PROGRAM MAIN
VAR
	bAllDone					: BOOL;
	bStopSequence				: BOOL;
	                    		
	nCase 						: INT;
	nMoveState				  	: ARRAY[GC.nNumMinMovers..GC.nNumMaxMovers] OF INT;
	                    		
	fbXtsEnvironment			: Tc3_XTS_Utility.FB_TcIoXtsEnvironment;
	                    		
	nForCounter					: UDINT;
	M,N,T,Tr					: UDINT;
	dynamics				    : INT;

//Status
	xSimulation					: BOOL := TRUE;
	SystemEnabled				: BOOL;

	IsMoverInBlockingArea		: BOOL;
	nActStopPos					: UINT := 1;
	Fp_error 					: Tc2_Standard.R_TRIG;
	FaultReset					: Tc2_Standard.R_TRIG;
	MoverStop 	AT%I* 			: BOOL;
    ResetSafetyLight AT%Q*      : BOOL;
	MoverStopDone AT%Q*			: BOOL;
	Info 		AT%Q*			: BOOL;
	Operating	AT%Q*			: BOOL;
	Process		AT%Q*			: BOOL;
	Fault		AT%Q*			: BOOL;
	Emergency	AT%Q*			: BOOL;
	                        	
	Voltage1	AT%I*			: UDINT;
	Voltage2	AT%I*			: UDINT;
	                        	
	TcRestart 					: Tc2_Utilities.TC_Restart;
	Restart 					: BOOL;
	busy 						: BOOL;
	fp_start 					: Tc2_Standard.R_TRIG;
	bStartSequence				: BOOL;
	                        	
	Horntimer 					: Tc2_Standard.TP; 
	R_trigHorn 					: Tc2_Standard.R_TRIG;

	StopTime 					: TIME := T#1S;
	StopTimer 					: ARRAY[GC.nNumMinMovers..GC.nNumMaxMovers] OF Tc2_Standard.TON;
	StartTimer 					: ARRAY[GC.nNumMinMovers..GC.nNumMaxMovers] OF BOOL;

	ArcLength 					: ARRAY[GC.nNumMinMovers..GC.nNumMaxMovers] OF LREAL;
	TrackPos					: ARRAY[GC.nNumMinMovers..GC.nNumMaxMovers] OF ARRAY[GC.nNumMinTracks..GC.nNumMaxTracks] OF Tc3_Physics.PositionXYC;
END_VAR

fbXtsEnvironment.Init(bExecute := TRUE);
//Cyclic
M_WritePlanarTrackConfig();
M_UpdateConfigurations();
IF xSimulation THEN
	SystemEnabled	:= TRUE;
ELSE
	SystemEnabled	:= (MoverStop (* SafetyOK *) AND NOT Fault);
END_IF

//Command Diverting to Magnet for any designated mover
DivertQueue();
HistoryDivertQueue(); // no removal
MergeQueue();

SwitchMagnet(SafetyPermIntlk := SystemEnabled,
			stSwitchConfig := GVL_General.stSwitchConfig);

Emergency :=  MoverStop;
ResetSafetyLight    := NOT MoverStop;

Operating := NOT  MoverStop;
R_trigHorn(clk := Voltage1> 10000 OR Voltage2 >10000);
Horntimer(in:= ( R_trigHorn.Q ) , PT:= T#2S,Q=> info);

IF nCase > 90 THEN
	Process := TRUE;
ELSE 
	Process := FALSE;	
END_IF

IF NOT fbXtsEnvironment.P_IsInitialized THEN
	RETURN;
END_IF

IF NOT MoverStop AND NOT MoverStopDone THEN
	FOR nForCounter:=1 TO nNumMovers DO
		aDynamics[nForCounter].SetValuesVADJ(V := stMoverConfig.MaxVelo, A := stMoverConfig.MaxAccel, D := stMoverConfig.MaxDecel, J := stMoverConfig.MaxJerk);
		nCase := 140;
		//fbPlanarMover[nForCounter].McPlanarMover.Halt(MoverFeedback[nForCounter], aDynamics[nForCounter]);
	END_FOR		
	MoverStopDone := TRUE;
ELSIF MoverStop THEN
	MoverStopDone := FALSE;
END_IF


TcRestart(
NETID:= '', 
RESTART:= Restart, 
TMOUT:=T#5S , 
BUSY=>busy , 
ERR=> , 
ERRID=> );


fp_start(CLK := bStartSequence);
IF fp_start.Q THEN
	nCase := 10;
	bStartSequence := FALSE;
END_IF

//IsMoverCommandedInShortcut := FALSE;
IsMoverInBlockingArea := FALSE;

	bAllDone:= TRUE;
FOR M := GC.nNumMinMovers TO nNumMovers DO///Movers
	StopTimer[M](in:=StartTimer[m],PT:=StopTime);
	GVL_Mc3.fbPlanarXtsMover[M].P_MoverId := M;
	GVL_Mc3.fbPlanarXtsMover[M].P_PlanarMover.MoverNumber	:= GVL_Mc3.fbPlanarXtsMover[M].nMoverId;
  GVL_Mc3.aiXpuXtsMover[M]  := fbXtsEnvironment.XpuTcIo(1).MoverTcIo(TO_UINT(M));
  fbPlanarXtsMover[M].iTcIoXtsXpuMover REF= GVL_Mc3.aiXpuXtsMover[M];
	fbPlanarXtsMover[M].Update();
	
	//MoverPos[M].SetValuesXYC(fbPlanarMover[M].McPlanarMover.MCTOPLC.SET.SetPos.x, fbPlanarMover[M].McPlanarMover.MCTOPLC.SET.SetPos.y,fbPlanarMover[M].McPlanarMover.MCTOPLC.SET.SetPos.c);
	
	TR := Tr+1;
	IF Tr = 4 THEN
		Tr :=1;
	END_IF
	{warning <'MoverPhysics does not work'>}
	ArcLength[M] :=GVL_Mc3.MC_Tracks[Tr].GetArcLengthClosestTo(GVL_Mc3.fbPlanarXtsMover[M].P_MoverPhysics);
	GVL_Mc3.MC_Tracks[Tr].GetPositionAt(ArcLength[M],TrackPos[M][Tr]);
	
//	IF ABS(GVL_Mc3.fbPlanarXtsMover[M].MoverPhysics.x - TrackPos[M][Tr].x) < 1 AND  ABS(fbPlanarXtsMover[M].MoverPhysics.y - TrackPos[M][Tr].y) < 1 THEN
// 		GVL_Mc3.fbPlanarXtsMover[M].P_XPlanarMover.MoverTrackNr := Tr;
//	END_IF	
	
//	IsMoverCommandedInShortcut := IsMoverCommandedInShortcut OR fbPlanarXtsMover[M].IsCommandedInShortcut;
//	IsMoverInBlockingArea := IsMoverInBlockingArea OR (GVL_Mc3.fbPlanarXtsMover[M].P_PlanarMover.TrackID = GVL_Mc3.MC_Tracks[E_TrackNum.main].MCTOPLC_STD.TrackOID AND 
//														IsBetween(value := GVL_Mc3.fbPlanarXtsMover[M].P_PlanarMover.MoverPos, 
//														minV := GVL_General.stSwitchConfig.fMagnetEntryPosn - GVL_General.stSwitchConfig.MagnetPosnComp, 
//														maxV :=  GVL_General.stSwitchConfig.fMagnetExitPosn + stSwitchConfig.MagnetPosnComp));
	MoverFeedback[M].Update();
	

	Fp_error(CLK := fbPlanarXtsMover[M].McPlanarMover.Error AND nCase = 100);
	IF Fp_error.Q THEN
		nCase := 140;
		Fault := TRUE;
//		bCmdMagnetOn := FALSE;
	END_IF
END_FOR

FOR T := GC.nNumMinTracks TO GC.nNumMaxTracks DO 
	MC_Tracks[T].Update();
	MC_Trackfeedback[T].Update();
END_FOR

CASE nCase OF
	10:
		Fault := FALSE;
		FOR nForCounter := 1 TO fbXtsEnvironment.XpuTcIo(1).GetPartCount() DO
			fbXtsEnvironment.XpuTcIo(1).PartTcIo(TO_UINT(nForCounter)).TriggerReset();
		END_FOR
		
		nCase := 20;

	20:
		FOR T := GC.nNumMinTracks TO GC.nNumMaxTracks DO 
			MC_Tracks[T].Enable(MC_Trackfeedback[T]);
		END_FOR
				nCase := 30;
		
		
	30: 
		IF MC_Trackfeedback[E_TrackNum.Big].Done AND MC_Trackfeedback[E_TrackNum.Main].Done AND MC_Trackfeedback[E_TrackNum.Small].Done THEN
			nCase := 35;
		END_IF
		
		
	35:
		FOR nForCounter:=GC.nNumMinMovers TO GVL_General.nNumMovers DO
			fbPlanarXtsMover[nForCounter].McPlanarMover.Reset(MoverFeedback[nForCounter]);
		END_FOR
		nCase := 36;	
		
		
	36:	
		bAllDone:=TRUE;
		FOR nForCounter:=GC.nNumMinMovers TO GVL_General.nNumMovers DO
			bAllDone:=bAllDone AND MoverFeedback[nForCounter].Done;
		END_FOR
		
		IF bAllDone THEN
			nCase := 40;
		END_IF
		
		
	40:
		FOR nForCounter:=GC.nNumMinMovers TO GVL_General.nNumMovers DO
			fbPlanarXtsMover[nForCounter].McPlanarMover.Enable(MoverFeedback[nForCounter]);
		END_FOR
		nCase := 50;
	
		
	50:
		bAllDone:=TRUE;
		FOR nForCounter:=GC.nNumMinMovers TO GVL_General.nNumMovers DO
			bAllDone:=bAllDone AND MoverFeedback[nForCounter].Done;
		END_FOR
		
		IF bAllDone THEN
			nCase := 60;
		END_IF

	//55:

	60:
		FOR nForCounter:=GC.nNumMinMovers TO GVL_General.nNumMovers DO
			IF nForCounter <= 9 THEN
				fbPlanarXtsMover[nForCounter].JoinTrack(MoverFeedback[nForCounter], GVL_Mc3.MC_Tracks[E_TrackNum.Big]);//   Mover[nForCounter].MoverTrackNr]);
			ELSE
				fbPlanarXtsMover[nForCounter].JoinTrack(MoverFeedback[nForCounter], GVL_Mc3.MC_Tracks[E_TrackNum.Main]);
			END_IF	
		END_FOR
		
		nCase := 70;
		
	70:
		bAllDone:=TRUE;
		FOR nForCounter:=GC.nNumMinMovers TO GVL_General.nNumMovers DO
			bAllDone:=bAllDone AND MoverFeedback[nForCounter].Done;
		END_FOR
		
		IF bAllDone THEN
			nCase := 80;
		END_IF
		
	80:	
		FOR nForCounter:=GC.nNumMinMovers TO GVL_General.nNumMovers DO
			nMoveState[nForCounter] := 0;
			aMoveOnTrackOptions[nForCounter].direction := MC_Direction.mcDirectionPositive;
			aMoveOnTrackOptions[nForCounter].gapMode := MC_GAP_MODE_ON_TRACK.Fast1D;
		END_FOR
		
		nCase := 100;

	100:

		FOR nForCounter:= GC.nNumMinMovers TO GVL_General.nNumMovers DO
			IF TrackSectors[nForCounter].SectorStatus[GC.SHORTCUT_HD_SECTION].MoverIsOnSector THEN
				//Increase dynamics on Inner Shortcut
				aDynamics[nForCounter].SetValuesVADJ(V := stMoverConfig.NormalVelo, A := stMoverConfig.MaxAccel, D := stMoverConfig.MaxDecel, J := stMoverConfig.MaxJerk);
//				aMoveOnTrackOptions[nForCounter].gap:= stMoverConfig.TightMoverGap;
			ELSE
				aDynamics[nForCounter].SetValuesVADJ(V := stMoverConfig.NormalVelo, A := stMoverConfig.NormalAccel, D := stMoverConfig.NormalDecel, J := stMoverConfig.NormalJerk);
				aMoveOnTrackOptions[nForCounter].gap:= stMoverConfig.NormalMoverGap;
			END_IF

			//Adjust the first mover parameters to induce a platoon
			aDynamics[GC.nNumMinMovers].SetValuesVADJ(V := stMoverConfig.NormalVelo-stMoverConfig.VeloComp, A := stMoverConfig.NormalAccel, D := stMoverConfig.NormalDecel, J := stMoverConfig.NormalJerk);

			// allow updating the config per the HMI, when it will not jeopardize the system
			IF NOT TrackSectors[nForCounter].SectorStatus[GC.MAG_TRIG_SECTOR_OPART_END].MoverIsOnSector AND NOT 
				TrackSectors[nForCounter].SectorStatus[GC.SHORTCUT_ENTRY_HALF_IPART].MoverIsOnSector THEN
				stSwitchConfig.SwitchModeInternal		:= 						stSwitchConfig.SwitchModeHMI;
			END_IF
			
//			IF TrackSectors[nForCounter].SectorStatus[GC.SHORTCUT_CALC_SECTOR_IPART].MoverEnteredSector.Q THEN
//				stSwitchStatus.ShuttleCountOnShortcut		:= stSwitchStatus.ShuttleCountOnShortcut + 1;
//			ELSIF TrackSectors[nForCounter].SectorStatus[GC.SHORTCUT_CALC_SECTOR_IPART].MoverExitedSector.Q THEN
//				stSwitchStatus.ShuttleCountOnShortcut		:= stSwitchStatus.ShuttleCountOnShortcut - 1;
//			END_IF
		
			TrackSectors[nForCounter](MoverIndex := nForCounter, XtsDataRef := fbPlanarXtsMover[nForCounter].P_XtsPositionInfo);
			HeadTrackSectors[nForCounter](MoverIndex := nForCounter, XtsDataRef := HeadExpMovers[nForCounter].stExpMoverStatus.XtsAdjustedData);
			TailTrackSectors[nForCounter](MoverIndex := nForCounter, XtsDataRef := TailExpMovers[nForCounter].stExpMoverStatus.XtsAdjustedData);			
			AllTrackSectors(TrackSectorsRef := GVL_Mc3.TrackSectors, HeadTrackSectorsRef := HeadTrackSectors, TailTrackSectorsRef := TailTrackSectors);
			
			HeadExpMovers[nForCounter](MoverRef := fbPlanarXtsMover[nForCounter]);
			TailExpMovers[nForCounter](MoverRef := fbPlanarXtsMover[nForCounter]);
			AllExpMovers(HeadMoversRef := HeadExpMovers, TailMoversRef := TailExpMovers);
			
			fbPlanarXtsMover[nForCounter]();
			
			CASE nMoveState[nForCounter] OF
				
				0: // Start-up/Init
					IF fbPlanarXtsMover[nForCounter].P_PlanarMover.TrackID = GVL_General.PlanarTrackOuterFinish THEN
						fbPlanarXtsMover[nForCounter].McPlanarMover.MoveOnTrack(commandFeedback := MoverFeedback[nForCounter],
																			targetTrack := GVL_Mc3.MC_Tracks[E_TrackNum.Big],
																			targetPositionOnTrack := GVL_Mc3.MC_Tracks[E_TrackNum.Big].GetLength()-stTrackGlobalConfig.TargetPosnBeforeTrackEnd,
																			constraint := aDynamics[nForCounter],
																			options := aMoveOnTrackOptions[nForCounter]);
						 nMoveState[nForCounter] 	:= 20;
					ELSIF fbPlanarXtsMover[nForCounter].P_PlanarMover.TrackID = GVL_General.PlanarTrackOuterStart THEN
						fbPlanarXtsMover[nForCounter].McPlanarMover.MoveOnTrack(commandFeedback := MoverFeedback[nForCounter],
																			targetTrack := GVL_Mc3.MC_Tracks[E_TrackNum.Main],
																			targetPositionOnTrack := GVL_Mc3.MC_Tracks[E_TrackNum.Main].GetLength()-stTrackGlobalConfig.TargetPosnBeforeTrackEnd,
																			constraint := aDynamics[nForCounter],
																			options := aMoveOnTrackOptions[nForCounter]);
						 nMoveState[nForCounter] 	:= 10;
					END_IF
					
				5: // In Recirc - from Big to Main Track
					fbPlanarXtsMover[nForCounter].McPlanarMover.MoveOnTrack(commandFeedback := MoverFeedback[nForCounter],
																		targetTrack := GVL_Mc3.MC_Tracks[E_TrackNum.Main],
																		targetPositionOnTrack := GVL_Mc3.MC_Tracks[E_TrackNum.Main].GetLength()-stTrackGlobalConfig.TargetPosnBeforeTrackEnd,
																		constraint := aDynamics[nForCounter],
																		options := aMoveOnTrackOptions[nForCounter]);
					 nMoveState[nForCounter] 	:= 10;

				10: //Trig state for decision to divert
					IF TrackSectors[nForCounter].afbSector[GC.MAG_TRIG_SECTOR_OPART_END].stSectorStatus.MoverEnteredSector.Q THEN
						GVL_General.stSwitchStatus.ShuttleCountAtDivertTrig		:= GVL_General.stSwitchStatus.ShuttleCountAtDivertTrig +1; //always MODing this; don't need to decrement
						TempMoverIndex	:= ((GVL_General.stSwitchStatus.ShuttleCountAtDivertTrig MOD GVL_General.stSwitchConfig.SwitchModeInternal.IntervalToDivert) +1); // capture the index
						DivertingMoverIndex := fbPlanarXtsMover[nForCounter].P_MoverId;
						AllTrackSectors.M_UpdateSectorCounts(SectorNr := GC.SHORTCUT_CALC_SECTOR_IPART);
						DivertQueue.M_UpdateAtTrig();
						nMoveState[nForCounter] 	:= 12;
					END_IF
					
				12:
					IF (stSwitchConfig.SwitchModeInternal.MaxAllowedDivertCount > 0) THEN
						IF (stSwitchStatus.ShuttleQueueCount > 0) AND NOT MagnetControlledByOtherMover THEN
							DivertQueue.RemoveObjFromBuffer();
							MagnetControlledByOtherMover	:= TRUE;
							// Divert Move command
							fbPlanarXtsMover[nForCounter].McPlanarMover.MoveOnTrack(commandFeedback := MoverFeedback[nForCounter],
																				targetTrack := GVL_Mc3.MC_Tracks[E_TrackNum.Small],
																				targetPositionOnTrack := (GVL_Mc3.MC_Tracks[E_TrackNum.Small].GetLength() - GC.SHUTTLE_LENGTH) / 2, // midpoint of shortcut
																				constraint := aDynamics[nForCounter],
																				options := aMoveOnTrackOptions[nForCounter]);
							nMoveState[nForCounter] 	:= 30; //Diverting Mover
						ELSIF NOT fbPlanarXtsMover[nForCounter].P_CmdDivert THEN
							nMoveState[nForCounter] 	:= 15;
						END_IF
					ELSIF TrackSectors[nForCounter].afbSector[GC.MAG_TRIG_SECTOR_OPART_END].stSectorStatus.MoverIsOnSector THEN
						 nMoveState[nForCounter] 	:= 15;
					END_IF
	
				15: // In Recirc - from Main to Big Track
					fbPlanarXtsMover[nForCounter].McPlanarMover.MoveOnTrack(commandFeedback := MoverFeedback[nForCounter],
																		targetTrack := GVL_Mc3.MC_Tracks[E_TrackNum.Big],
																		targetPositionOnTrack := GVL_Mc3.MC_Tracks[E_TrackNum.Big].GetLength()-stTrackGlobalConfig.TargetPosnBeforeTrackEnd,
																		constraint := aDynamics[nForCounter],
																		options := aMoveOnTrackOptions[nForCounter]);
					 nMoveState[nForCounter] 	:= 20;				
					
				20:
					IF TrackSectors[nForCounter].afbSector[GC.OUTER_BIGTRACK_END].stSectorStatus.MoverEnteredSector.Q THEN
						nMoveState[nForCounter]     := 5;
					END_IF				

				30: // Match the move command with the shuttle that is commanded to divert
					IF SwitchMagnet.P_PermIntlkOK THEN
						SwitchMagnet.M_EvaluateInlineCommands();
					END_IF
					IF NOT MagnetControlledByOtherMover THEN
						nMoveState[nForCounter] 	:= 40;
					END_IF
					
				40: // Confirm the shuttle is diverting
					IF TrackSectors[nForCounter].afbSector[GC.SHORTCUT_ENTRY_SECTOR_IPART].stSectorStatus.MoverExitedSector.Q THEN
						nMoveState[nForCounter] := 45;
					END_IF
			
				45: // Route through shortcut
					IF stTrackShortcutConfig.TestPowerMat THEN
						IF TrackSectors[nForCounter].afbSector[GC.LOAD_STOP_SECTOR_IPART].stSectorStatus.MoverEnteredSector.Q THEN
							nMoveState[nForCounter] := 70;
						END_IF
					ELSE		
						nMoveState[nForCounter] := 60;
					END_IF
					
				60: // Move to MergeWait Position
					fbPlanarXtsMover[nForCounter].McPlanarMover.MoveOnTrack(commandFeedback := MoverFeedback[nForCounter],
																		targetTrack := GVL_Mc3.MC_Tracks[E_TrackNum.Small],
																		targetPositionOnTrack := GVL_Mc3.MC_Tracks[E_TrackNum.Small].GetLength()-stTrackGlobalConfig.MergeWaitFinishDistance-stTrackGlobalConfig.MergeWaitAccelDistance,
																		constraint := aDynamics[nForCounter],
																		options := aMoveOnTrackOptions[nForCounter]);

					nMoveState[nForCounter] := 61;
					
				61:
				IF MoverFeedback[nForCounter].Done THEN
					nMoveState[nForCounter] := 62;
				END_IF
					
				62:// Permissive to Merge
					IF NOT AllTrackSectors.P_AMoverIsOnSector[GC.OUTER_MERGE_COLLISION] THEN
						nMoveState[nForCounter] := 63;
					END_IF

				63://Merge from Inner to Outer
						fbPlanarXtsMover[nForCounter].McPlanarMover.MoveOnTrack(commandFeedback := MoverFeedback[nForCounter],
																			targetTrack := GVL_Mc3.MC_Tracks[E_TrackNum.Small],
																			targetPositionOnTrack := GVL_Mc3.MC_Tracks[E_TrackNum.Small].GetLength()-stTrackGlobalConfig.TargetPosnBeforeTrackEnd,
																			constraint := aDynamics[nForCounter],
																			options := aMoveOnTrackOptions[nForCounter]);
						nMoveState[nForCounter] := 64;
				
				64: //Reset Command On Exit
						IF TrackSectors[nForCounter].afbSector[GC.INNER_MERGE_TO_FINISH].stSectorStatus.MoverIsOnSector THEN
							nMoveState[nForCounter] := 5;
						END_IF				

				70:
					IF MoverFeedback[nForCounter].Done THEN
						StartTimer[nForCounter] := TRUE;
						nMoveState[nForCounter] := 80;
					END_IF
					
				80:
					IF 	StopTimer[nForCounter].Q THEN
						StartTimer[nForCounter] := FALSE;
						nMoveState[nForCounter] := 60;	
					END_IF
				END_CASE
		
		END_FOR

		IF bStopSequence AND NOT(IsMoverInBlockingArea) THEN
			nCase := 110;
			bStopSequence := FALSE;
		END_IF
		110:
			N:= nNumMovers;
			FOR nForCounter:=1 TO nNumMovers DO		
				GVL_General.aStopPositions[nForCounter] := TO_LREAL(  fbXtsEnvironment.XpuTcIo(1).MoverTcIo(TO_UINT(N)).GetSimulatedStartUpPosition());
				N := N -1;
			END_FOR
			nCase := 120;
		
		120:	
			nActStopPos := UDINT_TO_UINT(GC.nNumMaxMovers-GVL_General.nNumMovers+1);
			FOR nForCounter:=1 TO nNumMovers DO
				aDynamics[nForCounter].SetValuesVADJ(V := stMoverConfig.StoppingVelo, A := stMoverConfig.NormalAccel, D := stMoverConfig.NormalDecel, J := stMoverConfig.NormalJerk);
				nMoveState[nForCounter] := 0;
				fbPlanarXtsMover[nForCounter].McPlanarMover.MoveOnTrack(MoverFeedback[nForCounter], GVL_Mc3.MC_Tracks[E_TrackNum.Main], 300, aDynamics[nForCounter],aMoveOnTrackOptions[nForCounter]);
			END_FOR

			nCase:= 130; 
		130:
			FOR nForCounter:=1 TO GC.nNumMaxMovers - (GVL_General.nNumMovers-GC.nNumMaxMovers)  DO
				CASE nMoveState[nForCounter] OF
					0:								
						
						IF GVL_Mc3.fbPlanarXtsMover[nForCounter].P_PlanarMover.MoverPos < 300 AND GVL_Mc3.fbPlanarXtsMover[nForCounter].P_PlanarMover.TrackID = GVL_Mc3.MC_Tracks[E_TrackNum.main].MCTOPLC_STD.TrackOID THEN
							aMoveOnTrackOptions[nForCounter].gap:= stMoverConfig.TightMoverGap;
							fbPlanarXtsMover[nForCounter].McPlanarMover.MoveOnTrack(commandFeedback := MoverFeedback[nForCounter],
																				targetTrack := GVL_Mc3.MC_Tracks[E_TrackNum.Main],
																				targetPositionOnTrack := aStopPositions[nActStopPos],
																				constraint := aDynamics[nForCounter],
																				options := aMoveOnTrackOptions[nForCounter]);									
							nActStopPos := nActStopPos + 1;
							nMoveState[nForCounter] := 10;
						END_IF
				END_CASE
			END_FOR
		
			bAllDone := TRUE;
			FOR nForCounter:=1 TO nNumMovers DO
				IF NOT(MoverFeedback[nForCounter].Done OR MoverFeedback[nForCounter].Error) THEN
					bAllDone := FALSE;
					EXIT;
				END_IF
			END_FOR
			
			IF bAllDone THEN
				nCase := 150;
			END_IF
		
		140:
			FOR nForCounter:=1 TO nNumMovers DO
				fbPlanarXtsMover[nForCounter].McPlanarMover.Halt(MoverFeedback[nForCounter], aDynamics[nForCounter]);
			END_FOR	
			
			nCase := 145;
			
		145:
			bAllDone := TRUE;
			FOR nForCounter:=1 TO nNumMovers DO
				IF NOT(MoverFeedback[nForCounter].Done OR MoverFeedback[nForCounter].Error) THEN
					bAllDone := FALSE;
					EXIT;
				END_IF
			END_FOR
			
			IF bAllDone THEN
				nCase := 150;
			END_IF
		
		//Disable
		150:
			FOR nForCounter:=1 TO nNumMovers DO
				fbPlanarXtsMover[nForCounter].McPlanarMover.Disable(MoverFeedback[nForCounter]);
			END_FOR
				
			nCase := 0;
END_CASE

FaultReset(CLK := MoverStop);

IF FaultReset.Q THEN
	Fault	:= FALSE;
END_IF

METHOD M_UpdateConfigurations
stTrackGlobalConfig.MergeWaitAccelDistance := 
F_PosnDisp(Accel := stMoverConfig.MaxAccel, 
								VeloFinal := stMoverConfig.NormalVelo, 
								VeloInit := 0);
END_METHOD

METHOD M_WritePlanarTrackConfig
stPlanarTrackConfig[E_TrackNum.Big].MCTrack				:= GVL_Mc3.MC_Tracks[E_TrackNum.Big].MCTOPLC_STD;
stPlanarTrackConfig[E_TrackNum.Small].MCTrack			:= GVL_Mc3.MC_Tracks[E_TrackNum.Small].MCTOPLC_STD;
stPlanarTrackConfig[E_TrackNum.Main].MCTrack			:= GVL_Mc3.MC_Tracks[E_TrackNum.Main].MCTOPLC_STD;
                                                    	
stPlanarTrackConfig[E_TrackNum.Big].TrackIndex			:= E_TrackNum.Big;
stPlanarTrackConfig[E_TrackNum.Small].TrackIndex		:= E_TrackNum.Small;
stPlanarTrackConfig[E_TrackNum.Main].TrackIndex			:= E_TrackNum.Main;
END_METHOD

END_PROGRAM

(* stored: Version 1.1.0.1
   POU MAIN: Id {66ade15a-bef8-4e71-a124-c2e5978c50eb}, SpecialFunc None
   Method M_UpdateConfigurations: Id {a2ceac5e-77e7-0f47-0d73-bb03330328f9}
   Method M_WritePlanarTrackConfig: Id {0295121c-55f9-0613-05f6-3ba76e5df670} *)
